// TIA Portal V19 export
TYPE "LEXCHANGETRAY_typeNgStrapControlNodeCommands"
TITLE = exchangeTray_typeNgStrapControlNodeCommands
// exchangeTray_typeNgStrapControlNodeCommands related values
// stored: Access Published
   STRUCT
      resetCount { ExternalAccessible := 'False'; ExternalVisible := 'False'; ExternalWritable := 'False'} : Bool;   // Reset count command
      resetError { ExternalAccessible := 'False'; ExternalVisible := 'False'; ExternalWritable := 'False'} : Bool;   // Reset error command
      raiseError { ExternalAccessible := 'False'; ExternalVisible := 'False'; ExternalWritable := 'False'} : Bool;   // Raise error command
      enable : Bool;
   END_STRUCT;
END_TYPE
